{attribute 'qualified_only'}
{attribute 'strict'}
{attribute 'to_string'}
TYPE E_ReqAction :
(
	NONE := 0, //Do Nothing
	INBOUND,
	OUTBOUND,
	DOCK_TB,
	UNOCK_TB
);
END_TYPE

(* stored: Version 1.1.0.1, ProductVersion 3.1.4024.12
   DUT E_ReqAction: Id {a67d854b-34ac-4a2d-be6e-be50abfd0cce} *)
